{attribute addProperty BoxType "EL3201-0030-0022"}
{attribute addProperty Id "RTDAT %I*RTD_B51B79FC8110.1250WcStateAT %I*WcState_F855686C1620InfoDataAT %I*InfoData_BC63D37F80100"}
{attribute addProperty CRC "1340698497"}
{attribute addProperty SizeInBites "177"}
{attribute addProperty SizeInBytes "22.125"}
TYPE EL3201_D2AFA856 :
STRUCT
	{attribute addProperty Name "RTD"}
	RTD : RTD_B51B79FC;
	{attribute addProperty Name "WcState"}
	WcState : WcState_F855686C;
	{attribute addProperty Name "InfoData"}
	InfoData : InfoData_BC63D37F;
END_STRUCT
END_TYPE

(* stored: Version 1.2.0.0, ProductVersion 3.1.4024.9
   DUT EL3201_D2AFA856: Id {89aba84e-d11b-48b6-8a56-93f0ec0360b3} *)
